// TIA Portal project "Project2" (V15.1)

(* hardware
DEVICE "S7300/ET200M station_1"  S7-300 station
   slot 0: "Rail_0"  Rail  6ES7 390-1***0-0AA0
   slot 2: "PLC_1"  CPU 312  6ES7 312-1AE14-0AB0  V3.3
      slot 0: "MPI interface_1"  MPI
*)

// ===== PLC "PLC_1"  CPU 312 =====

VAR_GLOBAL   // PLC tag table "Default tag table"
   "Radni" AT %I0.0 : Bool;   // 0 - nivo je ispod (nizak), 1 - nivo je iznad (visok)
   "Min" AT %I0.1 : Bool;   // 1 - OK, 0 - alarm (nizak nivo)
   "Reset alarma" AT %I0.2 : Bool;   // 1 - Reset
   "Pumpa" AT %Q4.0 : Bool;   // 1 - ON, 0 - OFF
   "R/A" AT %I0.4 : Bool;   // 0 - rucno, 1 - automatski
   "Start" AT %I0.5 : Bool;   // Start pumpe taster
   "Stop" AT %I0.6 : Bool;   // Stop pumpe taster
   "Rising Edge - Start" AT %M0.5 : Bool;
   "Rising Edge - Stop" AT %M0.6 : Bool;
   "Start / Stop Latch R" AT %M0.0 : Bool;
   "Start / Stop Latch A" AT %M0.1 : Bool;
   "Rucni rezim rada" AT %M1.0 : Bool;
   "Automatski rezim rada" AT %M1.1 : Bool;
   "Tag_1" AT %M0.2 : Bool;
   "Tag_2" AT %M2.0 : Bool;
   "Tag_3" AT %M2.1 : Bool;
   "Tag_4" AT %M2.5 : Bool;
   "Tag_5" AT %M2.4 : Bool;
   "Tag_6" AT %M2.7 : Bool;
   "Tag_7" AT %M3.0 : Bool;
END_VAR

DATA_BLOCK "Data_block_1"   // DB10
{ S7_Optimized_Access := 'FALSE' }
VERSION : 0.1
   VAR
      Alarm : Bool;   // Alarm
   END_VAR
BEGIN
END_DATA_BLOCK

FUNCTION "Mode" : Void   // FC1, LAD
{ S7_Optimized_Access := 'FALSE' }
VERSION : 0.1
   VAR_TEMP   // added for the SCL form of the ladder/FBD networks
      _w1 : Bool;
      _w2 : Bool;
   END_VAR
BEGIN

REGION Network 1: 1 - ON, 0 - OFF
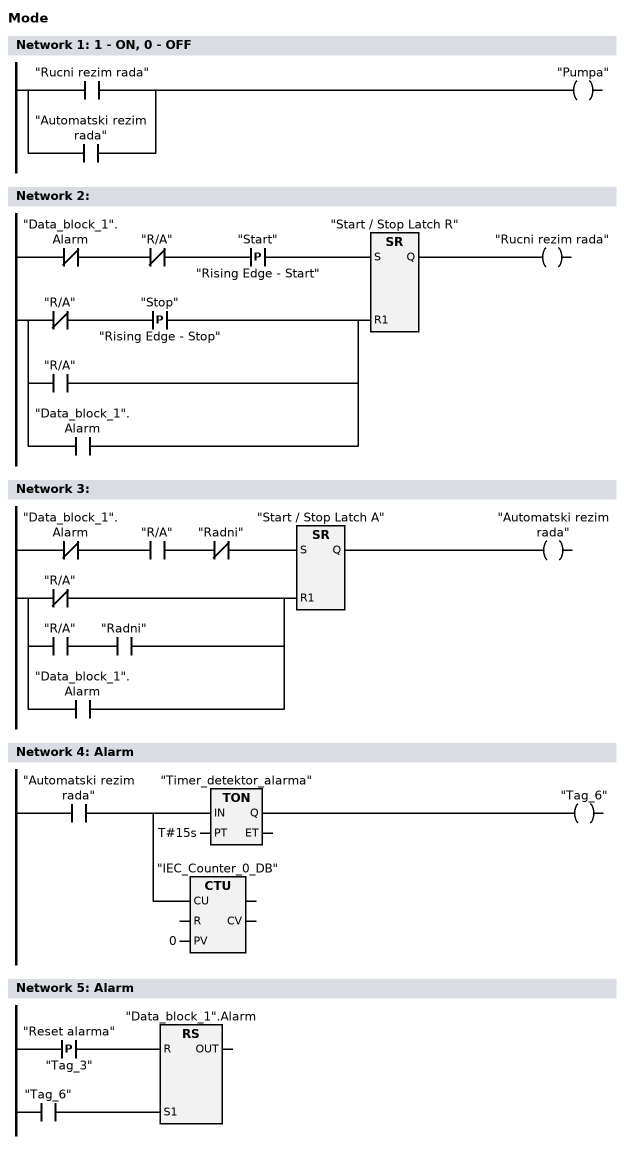
   RUNG wire#powerrail
      Contact( "Rucni rezim rada" )
      wire#w1
      Coil( "Pumpa" )
   END_RUNG
   RUNG wire#powerrail
      Contact( "Automatski rezim rada" )
   END_RUNG wire#w1
   // the same network as SCL:
   "Pumpa" := "Rucni rezim rada" OR "Automatski rezim rada";
END_REGION

REGION Network 2
   RUNG wire#powerrail
      I_Contact( "Data_block_1".Alarm )
      I_Contact( "R/A" )
      P_Contact(operand := "Start", bit := "Rising Edge - Start")
      S_SR(operand := "Start / Stop Latch R", r1 := wire#w1)
      Coil( "Rucni rezim rada" )
   END_RUNG
   RUNG wire#powerrail
      I_Contact( "R/A" )
      P_Contact(operand := "Stop", bit := "Rising Edge - Stop")
   END_RUNG wire#w1
   RUNG wire#powerrail
      Contact( "R/A" )
   END_RUNG wire#w1
   RUNG wire#powerrail
      Contact( "Data_block_1".Alarm )
   END_RUNG wire#w1
   // the same network as SCL:
   #_w1 := NOT "Data_block_1".Alarm AND NOT "R/A" AND "Start" AND NOT "Rising Edge - Start";   // rising edge of "Start"
   "Rising Edge - Start" := "Start";
   #_w2 := NOT "R/A" AND "Stop" AND NOT "Rising Edge - Stop";   // rising edge of "Stop"
   "Rising Edge - Stop" := "Stop";
   IF #_w1 THEN
       "Start / Stop Latch R" := TRUE;   // SR flip-flop
   END_IF;
   IF #_w2 OR "R/A" OR "Data_block_1".Alarm THEN "Start / Stop Latch R" := FALSE; END_IF;
   "Rucni rezim rada" := "Start / Stop Latch R";
END_REGION

REGION Network 3
   RUNG wire#powerrail
      I_Contact( "Data_block_1".Alarm )
      Contact( "R/A" )
      I_Contact( "Radni" )
      S_SR(operand := "Start / Stop Latch A", r1 := wire#w1)
      Coil( "Automatski rezim rada" )
   END_RUNG
   RUNG wire#powerrail
      I_Contact( "R/A" )
   END_RUNG wire#w1
   RUNG wire#powerrail
      Contact( "R/A" )
      Contact( "Radni" )
   END_RUNG wire#w1
   RUNG wire#powerrail
      Contact( "Data_block_1".Alarm )
   END_RUNG wire#w1
   // the same network as SCL:
   IF NOT "Data_block_1".Alarm AND "R/A" AND NOT "Radni" THEN
       "Start / Stop Latch A" := TRUE;   // SR flip-flop
   END_IF;
   IF NOT "R/A" OR ("R/A" AND "Radni") OR "Data_block_1".Alarm THEN "Start / Stop Latch A" := FALSE; END_IF;
   "Automatski rezim rada" := "Start / Stop Latch A";
END_REGION

REGION Network 4: Alarm
   "Timer_detektor_alarma".TON(IN := "Automatski rezim rada", PT := T#15s);
   "Tag_6" := "Timer_detektor_alarma".Q;
   "IEC_Counter_0_DB".CTU(CU := "Automatski rezim rada", PV := 0);
END_REGION

REGION Network 5: Alarm
   RUNG wire#powerrail
      P_Contact(operand := "Reset alarma", bit := "Tag_3")
      S_RS(operand := "Data_block_1".Alarm, s1 := wire#w1)
   END_RUNG
   RUNG wire#powerrail
      Contact( "Tag_6" )
   END_RUNG wire#w1
   // the same network as SCL:
   #_w1 := "Reset alarma" AND NOT "Tag_3";   // rising edge of "Reset alarma"
   "Tag_3" := "Reset alarma";
   IF #_w1 THEN
       "Data_block_1".Alarm := FALSE;   // RS flip-flop
   END_IF;
   IF "Tag_6" THEN "Data_block_1".Alarm := TRUE; END_IF;
END_REGION
END_FUNCTION

ORGANIZATION_BLOCK "Main"   // OB1, LAD
TITLE = "Main Program Sweep (Cycle)"
{ S7_Optimized_Access := 'FALSE' }
VERSION : 0.1
   VAR_TEMP
      OB1_EV_CLASS : Byte;   // Bits 0-3 = 1 (Coming event), Bits 4-7 = 1 (Event class 1)
      OB1_SCAN_1 : Byte;   // 1 (Cold restart scan 1 of OB 1), 3 (Scan 2-n of OB 1)
      OB1_PRIORITY : Byte;   // Priority of OB Execution
      OB1_OB_NUMBR : Byte;   // 1 (Organization block 1, OB1)
      OB1_RESERVED_1 : Byte;   // Reserved for system
      OB1_RESERVED_2 : Byte;   // Reserved for system
      OB1_PREV_CYCLE : Int;   // Cycle time of previous OB1 scan (milliseconds)
      OB1_MIN_CYCLE : Int;   // Minimum cycle time of OB1 (milliseconds)
      OB1_MAX_CYCLE : Int;   // Maximum cycle time of OB1 (milliseconds)
      OB1_DATE_TIME : Date_And_Time;   // Date and time OB1 started
   END_VAR
BEGIN

REGION Network 1
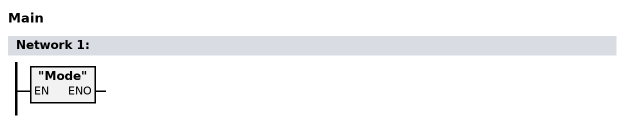
   RUNG wire#powerrail
      "Mode"()
   END_RUNG
   // the same network as SCL:
   "Mode"();
END_REGION
END_ORGANIZATION_BLOCK